INTERFACE ITF_NodeFactory

METHOD CreateNode : ITF_Node
VAR_INPUT
END_VAR
END_METHOD

METHOD DestroyNode : BOOL
VAR_INPUT
	Ptr		: PVOID;
END_VAR
END_METHOD

END_INTERFACE

(* stored: Version 1.1.0.1
   Itf ITF_NodeFactory: Id {fd4acf5c-33a2-4b48-8a41-f5b4f908e772}
   Method CreateNode: Id {a6cb453f-cc77-4858-9fe4-aa79b626eb32}
   Method DestroyNode: Id {acc9f66b-ee62-4043-b5a8-6b28b2c750fa} *)
